PROGRAM MAIN
VAR
	
END_VAR

GameEngine();

END_PROGRAM

(* stored: Version 1.1.0.1, ProductVersion 3.1.4024.4
   POU MAIN: Id {0fd8f3bb-2875-4327-87a4-a5acbddc9687}, SpecialFunc None *)
